FUNCTION_BLOCK FB_ControlSource_HMI_Machine EXTENDS FB_ControlSource_HMI
VAR_INPUT
END_VAR
VAR_OUTPUT
END_VAR
VAR
END_VAR

METHOD CyclicLogic
VAR_INPUT
END_VAR
SUPER^.CyclicLogic();

//Change the start permissive for the Machine 
MainPMLControl_Simplified.StartPermissive :=
    MainPMLControl_Standard.CurrentState = Tc3_PackML_V2.E_PMLState.ePMLState_Idle OR
    (MainPMLControl_Standard.CurrentState = Tc3_PackML_V2.E_PMLState.ePMLState_Held AND
    MAIN.ApicoSeed.Unwind.CurrentState = E_PMLState.ePMLState_Idle);
END_METHOD

END_FUNCTION_BLOCK

(* stored: Version 1.1.0.1, ProductVersion 3.1.4024.12
   POU FB_ControlSource_HMI_Machine: Id {b2bfe894-bd62-4bda-8587-75a7a69998f0}, SpecialFunc None
   Folder I_CyclicFB: Id {e68cdfcf-13d3-4757-96bc-cfed3982f6af}
   Method CyclicLogic: Id {b9558393-f6df-424b-bb06-aa52f94a69ed} *)
